Universal Robots PolyScope program: modbus_proba.urp

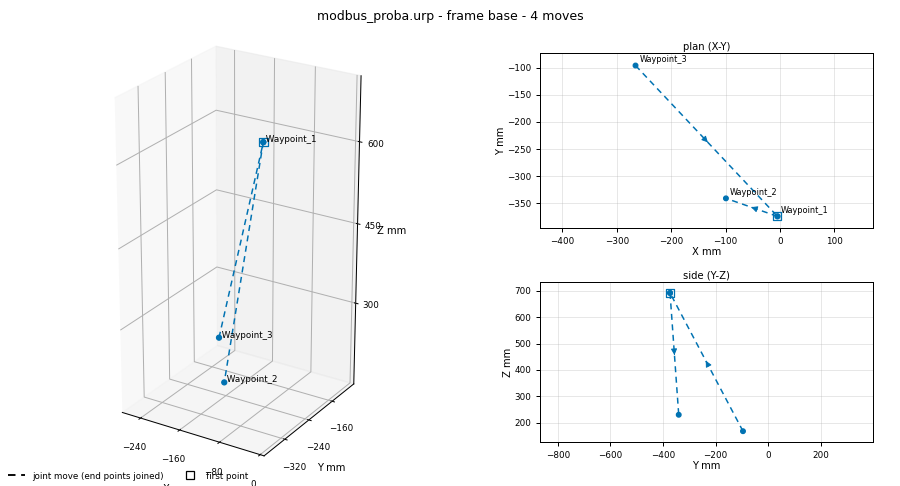
[picture p0: tool path of modbus_proba.urp in frame base, 4 of 5 moves have a stored position in this frame; points joined in program order, loops and branches not executed]
Program modbus_proba (installation=default directory=/programs/usbdisk createdIn=5.12.1.1101497 lastSavedIn=5.12.1.1101497 robotSerialNumber=20225300640)
Calibrated DH parameters: a=[-0.000125, -0.240482, -0.204397, 0.000169, -0.000135, 0]; d=[0.152056, 4.760815, 12.138494, -16.768367, 0.085457, 0.092357]; alpha=[1.570863, 0.008548, 0.003635, 1.571424, -1.571918, 0]; deltaTheta=[0, 0.167622, 0.124346, -0.291972, 0.000034, 0]
Robot Program (runOnlyOnce=false)
  'coordinates of the robot (in cm)'
  c_x := 0
  c_y := 0
  c_z := 0
  c_x := cx
  c_y := cy
  c_z := cz
  'We apply the signs to the abs values to reconstruct the coordinates'
  s_1 := s1
  s_2 := s2
  s_3 := s3
  c_x := (c_x/10) *(1-2*s_1)
  c_y := (c_y/10) *(1-2*s_2)
  c_z := (c_z/10) *(1-2*s_3)
  MoveJ speed 60 deg/s, acceleration 80 deg/s^2 (useActiveTCP=true) feature=Base
    Waypoint Waypoint_1: TCP in base x=-4.743 y=-373.657 z=692.583 mm, rx=-0.0132 ry=-2.2188 rz=2.2121 rad; joints [-0.002, -89.999, 0.002, -90.002, -0.001, 0.001] deg; TCP offset x=0.119 y=1.194 z=149.608 mm, rx=0 ry=0 rz=0 rad
  'Activation bit '
  Loop While (checkContinuously=false) expression=act≠1
    Wait Sleep waitTime=2
  Popup Warning (haltProgram=false message=Coordenades rebudes inputType=Text)
  Wait Sleep waitTime=0.01
  desti := p[c_x/100, c_y/100, c_z/100, 0.841, 3.028, -0.326]
  Popup Message (haltProgram=false inputType=Variable) variable=desti
  MoveJ speed 60 deg/s, acceleration 80 deg/s^2 (useActiveTCP=true) feature=Base
    Waypoint Waypoint_2: TCP in base x=-99.457 y=-340.562 z=229.498 mm, rx=0.0047 ry=3.0003 rz=-0.141 rad; joints [-89.798, -97.555, -64.497, -102.512, 98.076, 0.206] deg
    Wait Sleep waitTime=2
  MoveL speed 28 mm/s, acceleration 250 mm/s^2 (useActiveTCP=false) tcp=TCP; feature=Base
    Waypoint Waypoint (Variable): variable=desti
    Popup Message (haltProgram=false message=como lo ves inputType=Text)
    Wait Sleep waitTime=1
    MoveJ speed 60 deg/s, acceleration 80 deg/s^2 (useActiveTCP=true) feature=Base
      Waypoint Waypoint_3: TCP in base x=-265.692 y=-96.33 z=167.049 mm, rx=-3.1099 ry=-0.0533 rz=0.1236 rad; joints [-6.461, -105.626, 101.696, -90.868, -90.855, 81.067] deg
      Wait Sleep waitTime=0.5
      URCap Vacuum (Robotiq_Grippers, Robotiq Inc.) dataModel(Vacuum.Command.PumpAutoCloseDelayInMilliseconds=3000, Vacuum.Command.ShutOffDistance=5.0)
      Wait Sleep waitTime=2
      Waypoint Waypoint_4: TCP in base x=-4.683 y=-373.657 z=692.583 mm, rx=-0.0131 ry=-2.2188 rz=2.2121 rad; joints [-0.001, -90.002, -0.003, -90, 0, 0] deg
      URCap Vacuum (Robotiq_Grippers, Robotiq Inc.) dataModel(Vacuum.Command.Action=1, Vacuum.Command.PumpAutoCloseDelayInMilliseconds=3000, Vacuum.Command.ShutOffDistance=5.0)
    Wait Sleep waitTime=3
